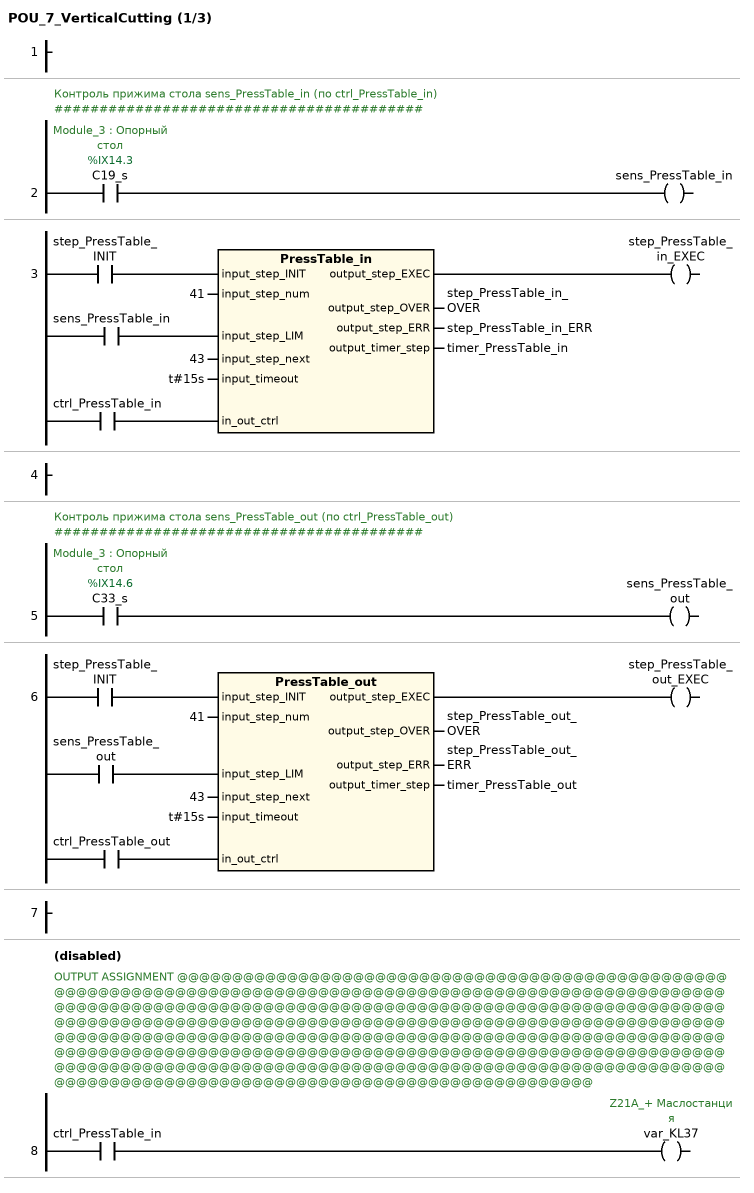
// NETWORK 1

// NETWORK 2
// Контроль прижима стола sens_PressTable_in (по ctrl_PressTable_in) #########################################
//   C19_s: Module_3 : Опорный стол | AT %IX14.3
sens_PressTable_in := C19_s;

// NETWORK 3
PressTable_in(input_step_INIT := step_PressTable_INIT, input_step_num := 41, input_step_LIM := sens_PressTable_in, input_step_next := 43, input_timeout := t#15s, in_out_ctrl := ctrl_PressTable_in, output_step_OVER => step_PressTable_in_OVER, output_step_ERR => step_PressTable_in_ERR, output_timer_step => timer_PressTable_in);
step_PressTable_in_EXEC := PressTable_in.output_step_EXEC;

// NETWORK 4

// NETWORK 5
// Контроль прижима стола sens_PressTable_out (по ctrl_PressTable_out) #########################################
//   C33_s: Module_3 : Опорный стол | AT %IX14.6
sens_PressTable_out := C33_s;

// NETWORK 6
PressTable_out(input_step_INIT := step_PressTable_INIT, input_step_num := 41, input_step_LIM := sens_PressTable_out, input_step_next := 43, input_timeout := t#15s, in_out_ctrl := ctrl_PressTable_out, output_step_OVER => step_PressTable_out_OVER, output_step_ERR => step_PressTable_out_ERR, output_timer_step => timer_PressTable_out);
step_PressTable_out_EXEC := PressTable_out.output_step_EXEC;

// NETWORK 7

// NETWORK 8 (disabled)
// OUTPUT ASSIGNMENT @@@@@@@@@@@@@@@@@@@@@@@@@@@@@@@@@@@@@@@@@@@@@@@@@@@@@@@@@@@@@@@@@@@@@@@@@@@@@@@@@@@@@@@@@@@@@@@@@@@@@@@@@@@@@@@@@@@@@@@@@@@@@@@@@@@@@@@@@@@@@@@@@@@@@@@@@@@@@@@@@@@@@@@@@@@@@@@@@@@@@@@@@@@@@@@@@@@@@@@@@@@@@@@@@@@@@@@@@@@@@@@@@@@@@@@@@@@@@@@@@@@@@@@@@@@@@@@@@@@@@@@@@@@@@@@@@@@@@@@@@@@@@@@@@@@@@@@@@@@@@@@@@@@@@@@@@@@@@@@@@@@@@@@@@@@@@@@@@@@@@@@@@@@@@@@@@@@@@@@@@@@@@@@@@@@@@@@@@@@@@@@@@@@@@@@@@@@@@@@@@@@@@@@@@@@@@@@@@@@@@@@@@@@@@@@@@@@@@@@@@@@@@@@@@@@@@@@@@@@@@@@@@
//   var_KL37: Z21A_+ Маслостанция
// var_KL37 := ctrl_PressTable_in;

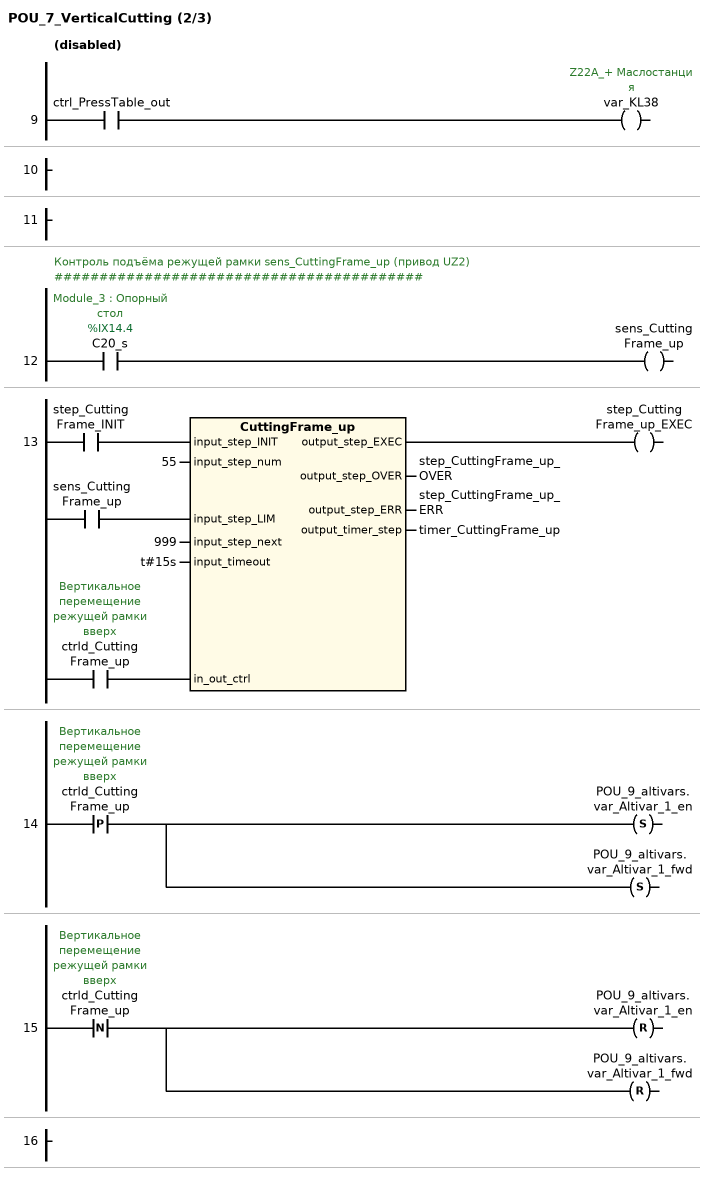
// NETWORK 9 (disabled)
//   var_KL38: Z22A_+ Маслостанция
// var_KL38 := ctrl_PressTable_out;

// NETWORK 10

// NETWORK 11

// NETWORK 12
// Контроль подъёма режущей рамки sens_CuttingFrame_up (привод UZ2) #########################################
//   C20_s: Module_3 : Опорный стол | AT %IX14.4
sens_CuttingFrame_up := C20_s;

// NETWORK 13
//   ctrld_CuttingFrame_up: Вертикальное перемещение режущей рамки вверх
CuttingFrame_up(input_step_INIT := step_CuttingFrame_INIT, input_step_num := 55, input_step_LIM := sens_CuttingFrame_up, input_step_next := 999, input_timeout := t#15s, in_out_ctrl := ctrld_CuttingFrame_up, output_step_OVER => step_CuttingFrame_up_OVER, output_step_ERR => step_CuttingFrame_up_ERR, output_timer_step => timer_CuttingFrame_up);
step_CuttingFrame_up_EXEC := CuttingFrame_up.output_step_EXEC;

// NETWORK 14
//   ctrld_CuttingFrame_up: Вертикальное перемещение режущей рамки вверх
_rt1(CLK := ctrld_CuttingFrame_up);
POU_9_altivars.var_Altivar_1_en S= _rt1.Q;
POU_9_altivars.var_Altivar_1_fwd S= _rt1.Q;

// NETWORK 15
//   ctrld_CuttingFrame_up: Вертикальное перемещение режущей рамки вверх
_ft1(CLK := ctrld_CuttingFrame_up);
POU_9_altivars.var_Altivar_1_en R= _ft1.Q;
POU_9_altivars.var_Altivar_1_fwd R= _ft1.Q;

// NETWORK 16

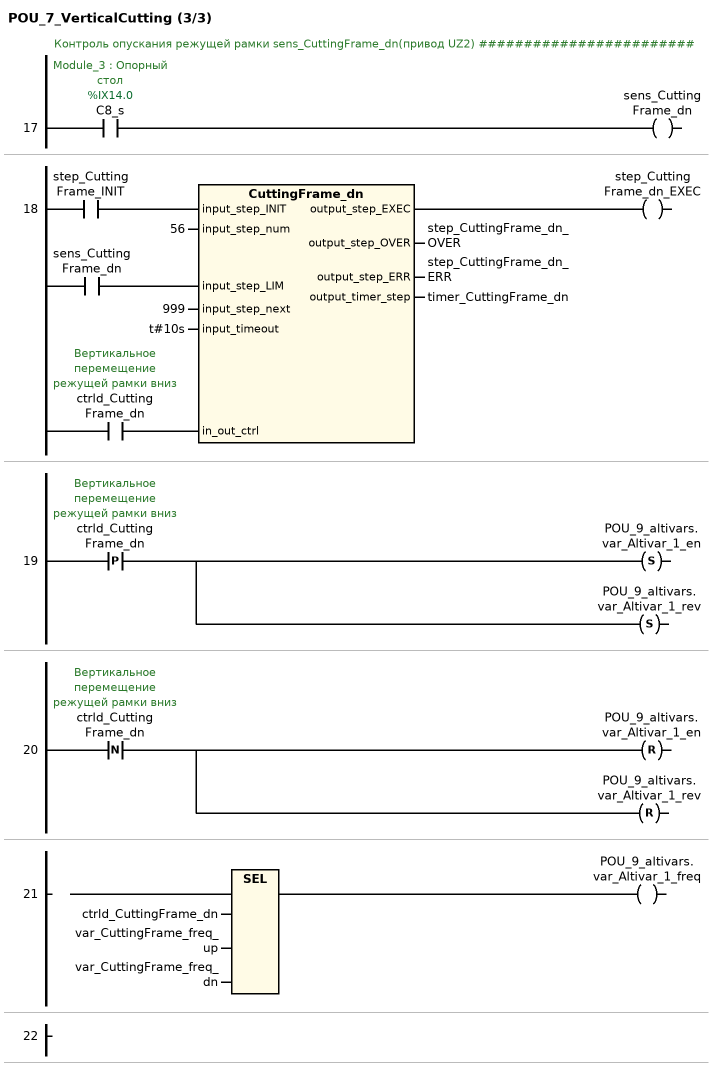
// NETWORK 17
// Контроль опускания режущей рамки sens_CuttingFrame_dn(привод UZ2) ########################
//   C8_s: Module_3 : Опорный стол | AT %IX14.0
sens_CuttingFrame_dn := C8_s;

// NETWORK 18
//   ctrld_CuttingFrame_dn: Вертикальное перемещение режущей рамки вниз
CuttingFrame_dn(input_step_INIT := step_CuttingFrame_INIT, input_step_num := 56, input_step_LIM := sens_CuttingFrame_dn, input_step_next := 999, input_timeout := t#10s, in_out_ctrl := ctrld_CuttingFrame_dn, output_step_OVER => step_CuttingFrame_dn_OVER, output_step_ERR => step_CuttingFrame_dn_ERR, output_timer_step => timer_CuttingFrame_dn);
step_CuttingFrame_dn_EXEC := CuttingFrame_dn.output_step_EXEC;

// NETWORK 19
//   ctrld_CuttingFrame_dn: Вертикальное перемещение режущей рамки вниз
_rt2(CLK := ctrld_CuttingFrame_dn);
POU_9_altivars.var_Altivar_1_en S= _rt2.Q;
POU_9_altivars.var_Altivar_1_rev S= _rt2.Q;

// NETWORK 20
//   ctrld_CuttingFrame_dn: Вертикальное перемещение режущей рамки вниз
_ft2(CLK := ctrld_CuttingFrame_dn);
POU_9_altivars.var_Altivar_1_en R= _ft2.Q;
POU_9_altivars.var_Altivar_1_rev R= _ft2.Q;

// NETWORK 21
//   ctrld_CuttingFrame_dn: Вертикальное перемещение режущей рамки вниз
POU_9_altivars.var_Altivar_1_freq := SEL(ctrld_CuttingFrame_dn, var_CuttingFrame_freq_up, var_CuttingFrame_freq_dn);

// NETWORK 22

END_PROGRAM

// MyController/Application/module_unites/PressTable_in
PROGRAM PressTable_in
VAR_INPUT
	input_step_INIT: BOOL;
	input_step_num: INT;
	input_step_LIM: BOOL;
	input_step_next: INT;
	input_timeout: TIME;
END_VAR

VAR_OUTPUT
	output_step_EXEC: BOOL;
	output_step_OVER: BOOL;
	output_step_ERR: BOOL;
	output_timer_step: TIME;
END_VAR
VAR_IN_OUT
	in_out_ctrl: BOOL;
END_VAR
VAR
	TON_step: TON;
	TON_step_res: BOOL;
	step_active: BOOL;
	TON_delay: TON;
	timer_delay: TIME;
	ton_delay_ok: BOOL;
END_VAR
VAR // added by the converter: edge detectors and wires of the graphical bodies
    _rt1, _rt2, _rt3, _rt4, _rt5, _rt6, _rt7 : R_TRIG;
    _w1, _w2 : BOOL;
    _ft1 : F_TRIG;
END_VAR

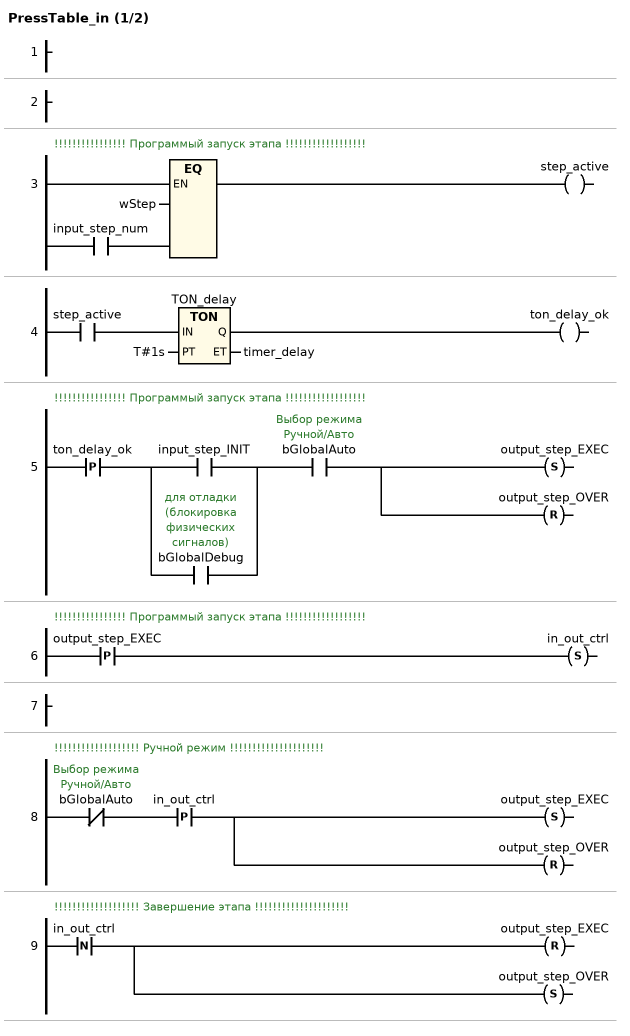
// NETWORK 1

// NETWORK 2

// NETWORK 3
// !!!!!!!!!!!!!!!! Программый запуск этапа !!!!!!!!!!!!!!!!!!
step_active := wStep = input_step_num;

// NETWORK 4
TON_delay(IN := step_active, PT := T#1s, ET => timer_delay); // TON
ton_delay_ok := TON_delay.Q;

// NETWORK 5
// !!!!!!!!!!!!!!!! Программый запуск этапа !!!!!!!!!!!!!!!!!!
//   bGlobalDebug: для отладки (блокировка физических сигналов)
//   bGlobalAuto: Выбор режима Ручной/Авто
_rt1(CLK := ton_delay_ok);
_w1 := _rt1.Q AND (input_step_INIT OR bGlobalDebug) AND bGlobalAuto;
output_step_EXEC S= _w1;
output_step_OVER R= _w1;

// NETWORK 6
// !!!!!!!!!!!!!!!! Программый запуск этапа !!!!!!!!!!!!!!!!!!
_rt2(CLK := output_step_EXEC);
in_out_ctrl S= _rt2.Q;

// NETWORK 7

// NETWORK 8
// !!!!!!!!!!!!!!!!!!! Ручной режим !!!!!!!!!!!!!!!!!!!!!
//   bGlobalAuto: Выбор режима Ручной/Авто
_rt3(CLK := in_out_ctrl);
_w2 := NOT bGlobalAuto AND _rt3.Q;
output_step_EXEC S= _w2;
output_step_OVER R= _w2;

// NETWORK 9
// !!!!!!!!!!!!!!!!!!! Завершение этапа !!!!!!!!!!!!!!!!!!!!!
_ft1(CLK := in_out_ctrl);
output_step_EXEC R= _ft1.Q;
output_step_OVER S= _ft1.Q;

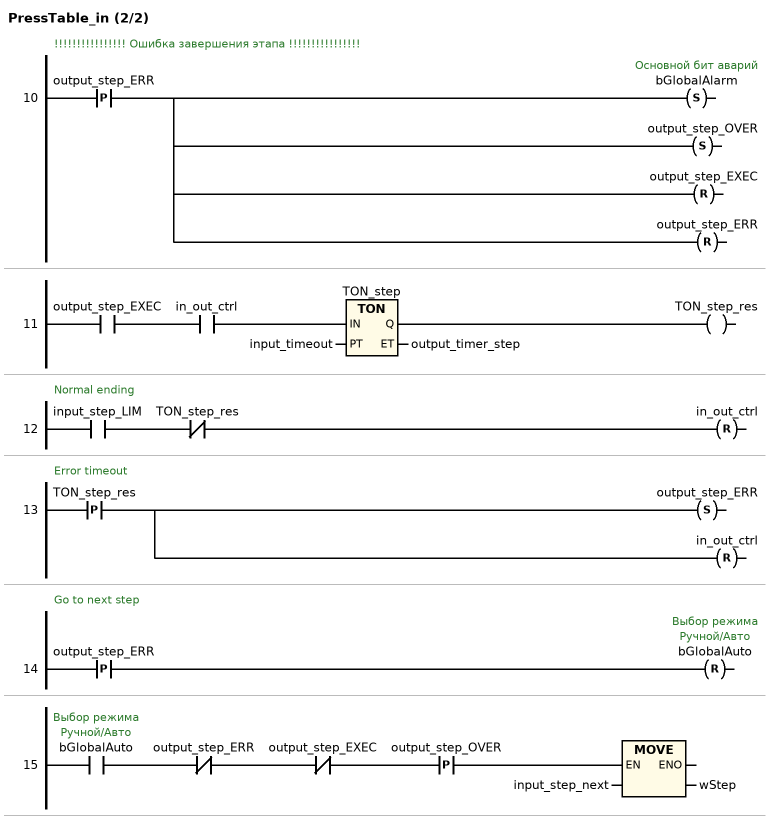
// NETWORK 10
// !!!!!!!!!!!!!!!! Ошибка завершения этапа !!!!!!!!!!!!!!!!
//   bGlobalAlarm: Основной бит аварий
_rt4(CLK := output_step_ERR);
bGlobalAlarm S= _rt4.Q;
output_step_OVER S= _rt4.Q;
output_step_EXEC R= _rt4.Q;
output_step_ERR R= _rt4.Q;

// NETWORK 11
TON_step(IN := output_step_EXEC AND in_out_ctrl, PT := input_timeout, ET => output_timer_step); // TON
TON_step_res := TON_step.Q;

// NETWORK 12
// Normal ending
in_out_ctrl R= input_step_LIM AND NOT TON_step_res;

// NETWORK 13
// Error timeout
_rt5(CLK := TON_step_res);
output_step_ERR S= _rt5.Q;
in_out_ctrl R= _rt5.Q;

// NETWORK 14
// Go to next step
//   bGlobalAuto: Выбор режима Ручной/Авто
_rt6(CLK := output_step_ERR);
bGlobalAuto R= _rt6.Q;

// NETWORK 15
//   bGlobalAuto: Выбор режима Ручной/Авто
_rt7(CLK := output_step_OVER);
IF bGlobalAuto AND NOT output_step_ERR AND NOT output_step_EXEC AND _rt7.Q THEN wStep := input_step_next; END_IF

END_PROGRAM

// MyController/Application/module_unites/PressTable_out
PROGRAM PressTable_out
VAR_INPUT
	input_step_INIT: BOOL;
	input_step_num: INT;
	input_step_LIM: BOOL;
	input_step_next: INT;
	input_timeout: TIME;
END_VAR

VAR_OUTPUT
	output_step_EXEC: BOOL;
	output_step_OVER: BOOL;
	output_step_ERR: BOOL;
	output_timer_step: TIME;
END_VAR
VAR_IN_OUT
	in_out_ctrl: BOOL;
END_VAR
VAR
	TON_step: TON;
	TON_step_res: BOOL;
	step_active: BOOL;
	TON_delay: TON;
	timer_delay: TIME;
	ton_delay_ok: BOOL;
END_VAR
VAR // added by the converter: edge detectors and wires of the graphical bodies
    _rt1, _rt2, _rt3, _rt4, _rt5, _rt6, _rt7 : R_TRIG;
    _w1, _w2 : BOOL;
    _ft1 : F_TRIG;
END_VAR

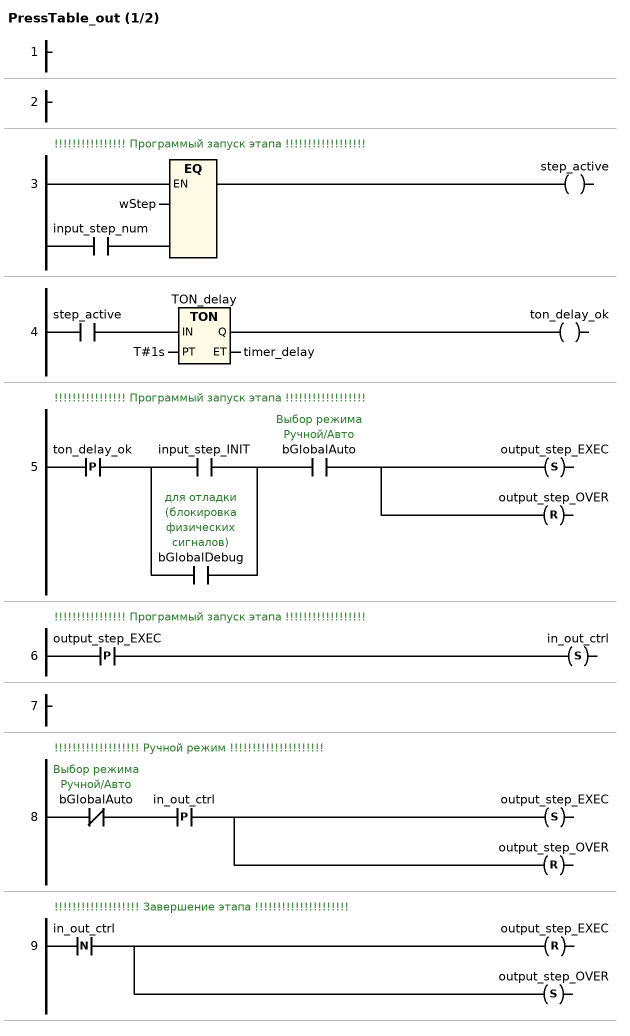
// NETWORK 1

// NETWORK 2

// NETWORK 3
// !!!!!!!!!!!!!!!! Программый запуск этапа !!!!!!!!!!!!!!!!!!
step_active := wStep = input_step_num;

// NETWORK 4
TON_delay(IN := step_active, PT := T#1s, ET => timer_delay); // TON
ton_delay_ok := TON_delay.Q;

// NETWORK 5
// !!!!!!!!!!!!!!!! Программый запуск этапа !!!!!!!!!!!!!!!!!!
//   bGlobalDebug: для отладки (блокировка физических сигналов)
//   bGlobalAuto: Выбор режима Ручной/Авто
_rt1(CLK := ton_delay_ok);
_w1 := _rt1.Q AND (input_step_INIT OR bGlobalDebug) AND bGlobalAuto;
output_step_EXEC S= _w1;
output_step_OVER R= _w1;

// NETWORK 6
// !!!!!!!!!!!!!!!! Программый запуск этапа !!!!!!!!!!!!!!!!!!
_rt2(CLK := output_step_EXEC);
in_out_ctrl S= _rt2.Q;

// NETWORK 7

// NETWORK 8
// !!!!!!!!!!!!!!!!!!! Ручной режим !!!!!!!!!!!!!!!!!!!!!
//   bGlobalAuto: Выбор режима Ручной/Авто
_rt3(CLK := in_out_ctrl);
_w2 := NOT bGlobalAuto AND _rt3.Q;
output_step_EXEC S= _w2;
output_step_OVER R= _w2;

// NETWORK 9
// !!!!!!!!!!!!!!!!!!! Завершение этапа !!!!!!!!!!!!!!!!!!!!!
_ft1(CLK := in_out_ctrl);
output_step_EXEC R= _ft1.Q;
output_step_OVER S= _ft1.Q;

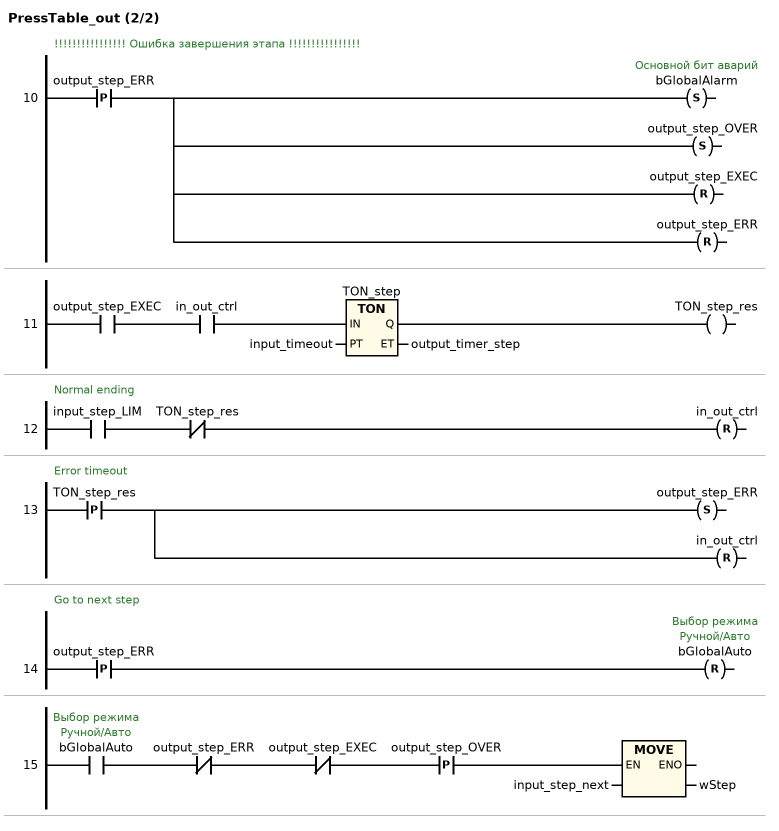
// NETWORK 10
// !!!!!!!!!!!!!!!! Ошибка завершения этапа !!!!!!!!!!!!!!!!
//   bGlobalAlarm: Основной бит аварий
_rt4(CLK := output_step_ERR);
bGlobalAlarm S= _rt4.Q;
output_step_OVER S= _rt4.Q;
output_step_EXEC R= _rt4.Q;
output_step_ERR R= _rt4.Q;

// NETWORK 11
TON_step(IN := output_step_EXEC AND in_out_ctrl, PT := input_timeout, ET => output_timer_step); // TON
TON_step_res := TON_step.Q;

// NETWORK 12
// Normal ending
in_out_ctrl R= input_step_LIM AND NOT TON_step_res;

// NETWORK 13
// Error timeout
_rt5(CLK := TON_step_res);
output_step_ERR S= _rt5.Q;
in_out_ctrl R= _rt5.Q;

// NETWORK 14
// Go to next step
//   bGlobalAuto: Выбор режима Ручной/Авто
_rt6(CLK := output_step_ERR);
bGlobalAuto R= _rt6.Q;

// NETWORK 15
//   bGlobalAuto: Выбор режима Ручной/Авто
_rt7(CLK := output_step_OVER);
IF bGlobalAuto AND NOT output_step_ERR AND NOT output_step_EXEC AND _rt7.Q THEN wStep := input_step_next; END_IF

END_PROGRAM

// MyController/Application/module_unites/CuttingFrame_up
PROGRAM CuttingFrame_up
VAR_INPUT
	input_step_INIT: BOOL;
	input_step_num: INT;
	input_step_LIM: BOOL;
	input_step_next: INT;
	input_timeout: TIME;
END_VAR

VAR_OUTPUT
	output_step_EXEC: BOOL;
	output_step_OVER: BOOL;
	output_step_ERR: BOOL;
	output_timer_step: TIME;
END_VAR
VAR_IN_OUT
	in_out_ctrl: BOOL;
END_VAR
VAR
	TON_step: TON;
	TON_step_res: BOOL;
	step_active: BOOL;
	TON_delay: TON;
	timer_delay: TIME;
	ton_delay_ok: BOOL;
END_VAR
VAR // added by the converter: edge detectors and wires of the graphical bodies
    _rt1, _rt2, _rt3, _rt4, _rt5, _rt6, _rt7 : R_TRIG;
    _w1, _w2 : BOOL;
    _ft1 : F_TRIG;
END_VAR

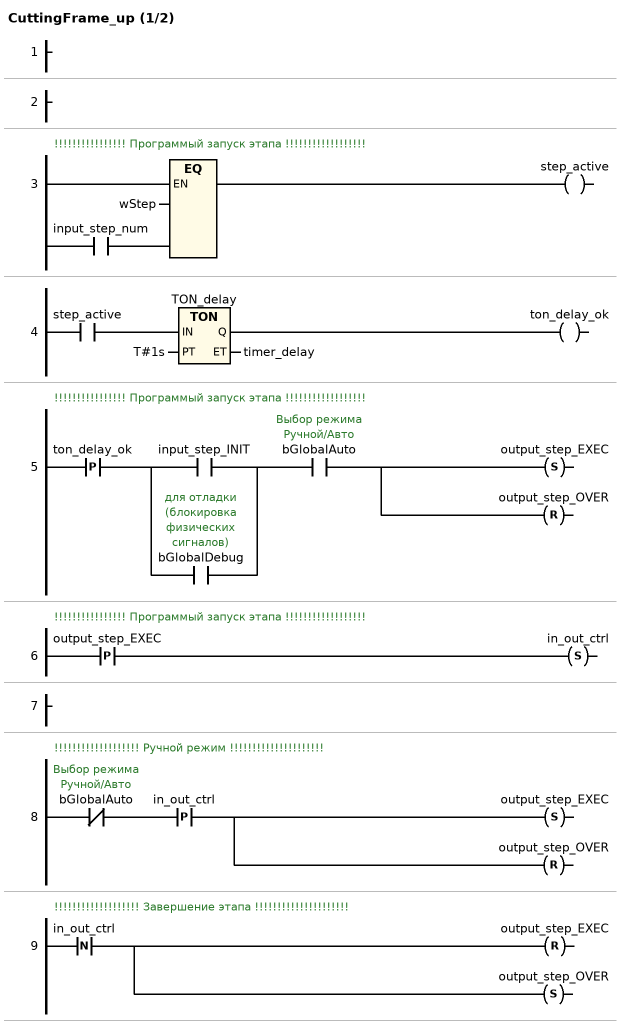
// NETWORK 1

// NETWORK 2

// NETWORK 3
// !!!!!!!!!!!!!!!! Программый запуск этапа !!!!!!!!!!!!!!!!!!
step_active := wStep = input_step_num;

// NETWORK 4
TON_delay(IN := step_active, PT := T#1s, ET => timer_delay); // TON
ton_delay_ok := TON_delay.Q;

// NETWORK 5
// !!!!!!!!!!!!!!!! Программый запуск этапа !!!!!!!!!!!!!!!!!!
//   bGlobalDebug: для отладки (блокировка физических сигналов)
//   bGlobalAuto: Выбор режима Ручной/Авто
_rt1(CLK := ton_delay_ok);
_w1 := _rt1.Q AND (input_step_INIT OR bGlobalDebug) AND bGlobalAuto;
output_step_EXEC S= _w1;
output_step_OVER R= _w1;

// NETWORK 6
// !!!!!!!!!!!!!!!! Программый запуск этапа !!!!!!!!!!!!!!!!!!
_rt2(CLK := output_step_EXEC);
in_out_ctrl S= _rt2.Q;

// NETWORK 7

// NETWORK 8
// !!!!!!!!!!!!!!!!!!! Ручной режим !!!!!!!!!!!!!!!!!!!!!
//   bGlobalAuto: Выбор режима Ручной/Авто
_rt3(CLK := in_out_ctrl);
_w2 := NOT bGlobalAuto AND _rt3.Q;
output_step_EXEC S= _w2;
output_step_OVER R= _w2;

// NETWORK 9
// !!!!!!!!!!!!!!!!!!! Завершение этапа !!!!!!!!!!!!!!!!!!!!!
_ft1(CLK := in_out_ctrl);
output_step_EXEC R= _ft1.Q;
output_step_OVER S= _ft1.Q;

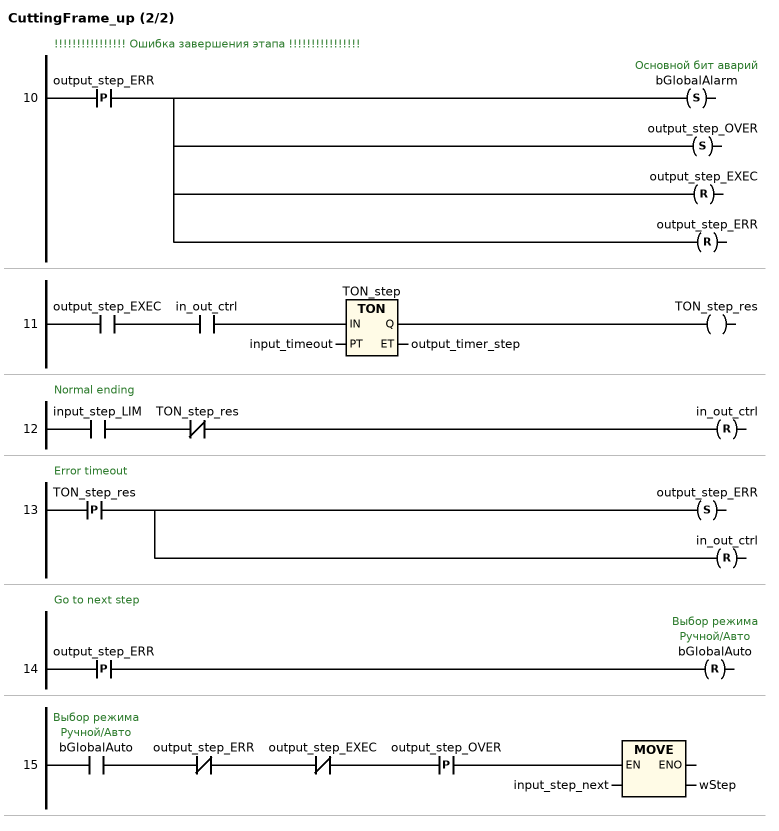
// NETWORK 10
// !!!!!!!!!!!!!!!! Ошибка завершения этапа !!!!!!!!!!!!!!!!
//   bGlobalAlarm: Основной бит аварий
_rt4(CLK := output_step_ERR);
bGlobalAlarm S= _rt4.Q;
output_step_OVER S= _rt4.Q;
output_step_EXEC R= _rt4.Q;
output_step_ERR R= _rt4.Q;

// NETWORK 11
TON_step(IN := output_step_EXEC AND in_out_ctrl, PT := input_timeout, ET => output_timer_step); // TON
TON_step_res := TON_step.Q;

// NETWORK 12
// Normal ending
in_out_ctrl R= input_step_LIM AND NOT TON_step_res;

// NETWORK 13
// Error timeout
_rt5(CLK := TON_step_res);
output_step_ERR S= _rt5.Q;
in_out_ctrl R= _rt5.Q;

// NETWORK 14
// Go to next step
//   bGlobalAuto: Выбор режима Ручной/Авто
_rt6(CLK := output_step_ERR);
bGlobalAuto R= _rt6.Q;

// NETWORK 15
//   bGlobalAuto: Выбор режима Ручной/Авто
_rt7(CLK := output_step_OVER);
IF bGlobalAuto AND NOT output_step_ERR AND NOT output_step_EXEC AND _rt7.Q THEN wStep := input_step_next; END_IF

END_PROGRAM

// MyController/Application/module_unites/CuttingFrame_dn
PROGRAM CuttingFrame_dn
VAR_INPUT
	input_step_INIT: BOOL;
	input_step_num: INT;
	input_step_LIM: BOOL;
	input_step_next: INT;
	input_timeout: TIME;
END_VAR

VAR_OUTPUT
	output_step_EXEC: BOOL;
	output_step_OVER: BOOL;
	output_step_ERR: BOOL;
	output_timer_step: TIME;
END_VAR
VAR_IN_OUT
	in_out_ctrl: BOOL;
END_VAR
VAR
	TON_step: TON;
	TON_step_res: BOOL;
	step_active: BOOL;
	TON_delay: TON;
	timer_delay: TIME;
	ton_delay_ok: BOOL;
END_VAR
VAR // added by the converter: edge detectors and wires of the graphical bodies
    _rt1, _rt2, _rt3, _rt4, _rt5, _rt6, _rt7 : R_TRIG;
    _w1, _w2 : BOOL;
    _ft1 : F_TRIG;
END_VAR

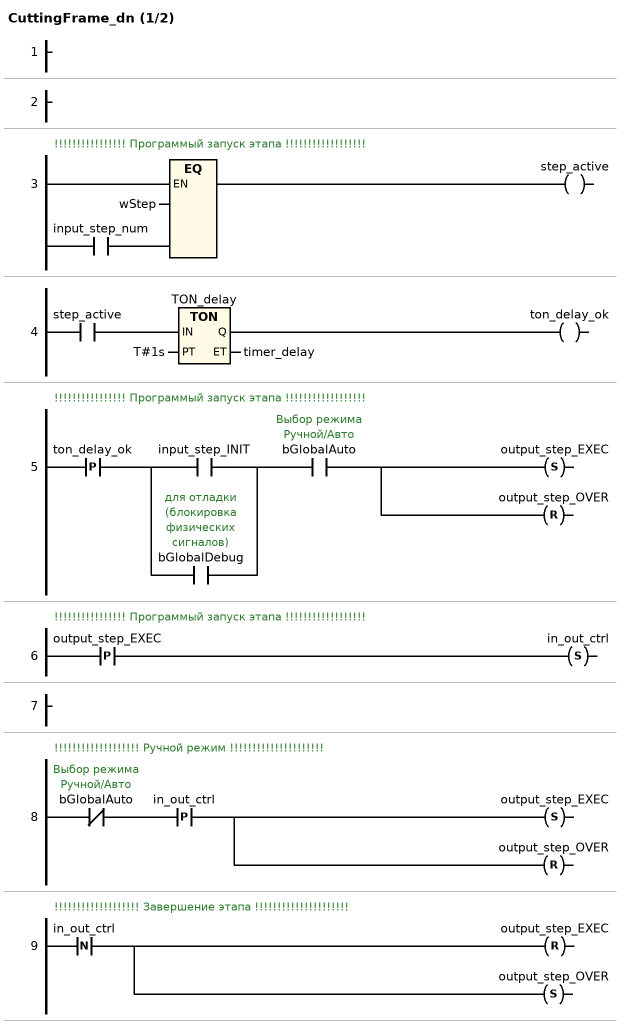
// NETWORK 1

// NETWORK 2

// NETWORK 3
// !!!!!!!!!!!!!!!! Программый запуск этапа !!!!!!!!!!!!!!!!!!
step_active := wStep = input_step_num;

// NETWORK 4
TON_delay(IN := step_active, PT := T#1s, ET => timer_delay); // TON
ton_delay_ok := TON_delay.Q;

// NETWORK 5
// !!!!!!!!!!!!!!!! Программый запуск этапа !!!!!!!!!!!!!!!!!!
//   bGlobalDebug: для отладки (блокировка физических сигналов)
//   bGlobalAuto: Выбор режима Ручной/Авто
_rt1(CLK := ton_delay_ok);
_w1 := _rt1.Q AND (input_step_INIT OR bGlobalDebug) AND bGlobalAuto;
output_step_EXEC S= _w1;
output_step_OVER R= _w1;

// NETWORK 6
// !!!!!!!!!!!!!!!! Программый запуск этапа !!!!!!!!!!!!!!!!!!
_rt2(CLK := output_step_EXEC);
in_out_ctrl S= _rt2.Q;

// NETWORK 7

// NETWORK 8
// !!!!!!!!!!!!!!!!!!! Ручной режим !!!!!!!!!!!!!!!!!!!!!
//   bGlobalAuto: Выбор режима Ручной/Авто
_rt3(CLK := in_out_ctrl);
_w2 := NOT bGlobalAuto AND _rt3.Q;
output_step_EXEC S= _w2;
output_step_OVER R= _w2;

// NETWORK 9
// !!!!!!!!!!!!!!!!!!! Завершение этапа !!!!!!!!!!!!!!!!!!!!!
_ft1(CLK := in_out_ctrl);
output_step_EXEC R= _ft1.Q;
output_step_OVER S= _ft1.Q;

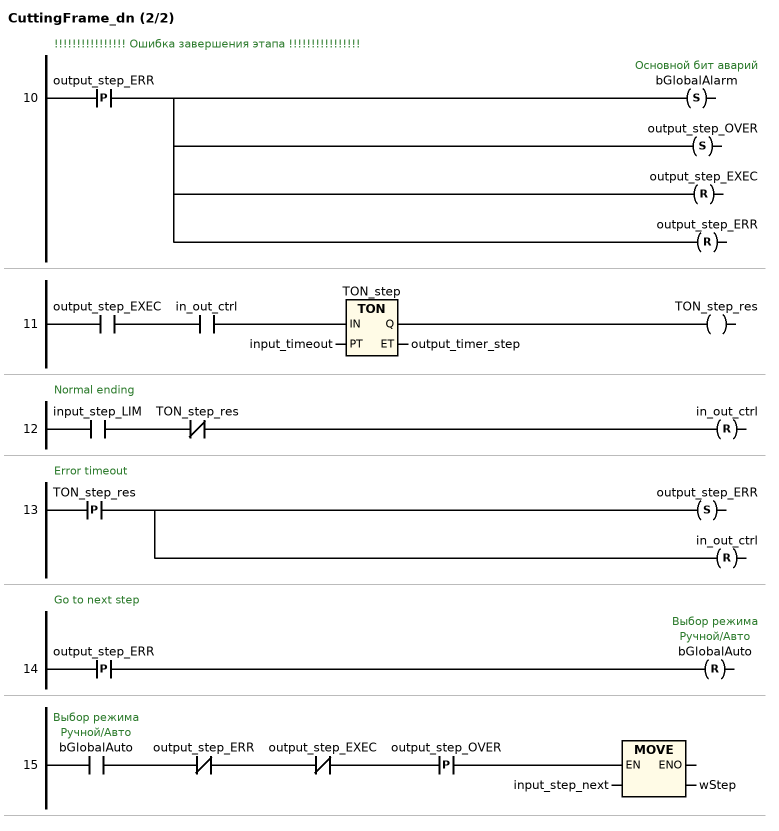
// NETWORK 10
// !!!!!!!!!!!!!!!! Ошибка завершения этапа !!!!!!!!!!!!!!!!
//   bGlobalAlarm: Основной бит аварий
_rt4(CLK := output_step_ERR);
bGlobalAlarm S= _rt4.Q;
output_step_OVER S= _rt4.Q;
output_step_EXEC R= _rt4.Q;
output_step_ERR R= _rt4.Q;

// NETWORK 11
TON_step(IN := output_step_EXEC AND in_out_ctrl, PT := input_timeout, ET => output_timer_step); // TON
TON_step_res := TON_step.Q;

// NETWORK 12
// Normal ending
in_out_ctrl R= input_step_LIM AND NOT TON_step_res;

// NETWORK 13
// Error timeout
_rt5(CLK := TON_step_res);
output_step_ERR S= _rt5.Q;
in_out_ctrl R= _rt5.Q;

// NETWORK 14
// Go to next step
//   bGlobalAuto: Выбор режима Ручной/Авто
_rt6(CLK := output_step_ERR);
bGlobalAuto R= _rt6.Q;

// NETWORK 15
//   bGlobalAuto: Выбор режима Ручной/Авто
_rt7(CLK := output_step_OVER);
IF bGlobalAuto AND NOT output_step_ERR AND NOT output_step_EXEC AND _rt7.Q THEN wStep := input_step_next; END_IF

END_PROGRAM

// MyController/Application/POU_5_Oprokidyvanie
PROGRAM POU_5_Oprokidyvanie
VAR
	sens_TakeTable_in: BOOL;
	ctrl_TakeTable_in: BOOL;
	step_TakeTable_INIT: BOOL := TRUE;
	step_TakeTable_in_EXEC: BOOL;
	step_TakeTable_in_OVER: BOOL;
	step_TakeTable_in_ERR: BOOL;
	timer_TakeTable_in: TIME;
	ctrl_TakeTable_out: BOOL;
	sens_TakeTable_out: BOOL;
	step_TakeTable_out_EXEC: BOOL;
	step_TakeTable_out_OVER: BOOL;
	step_TakeTable_out_ERR: BOOL;
	timer_TakeTable_out: TIME;
	ctrl_MoveTipper_in: BOOL;
	sens_MoveTipper_in: BOOL;
	step_MoveTipper_INIT: BOOL := TRUE;
	step_MoveTipper_in_EXEC: BOOL;
	step_MoveTipper_in_OVER: BOOL;
	step_MoveTipper_in_ERR: BOOL;
	timer_MoveTipper_in: TIME;
	ctrl_MoveTipper_out: BOOL;
	sens_MoveTipper_out: BOOL;
	step_MoveTipper_out_EXEC: BOOL;
	step_MoveTipper_out_OVER: BOOL;
	step_MoveTipper_out_ERR: BOOL;
	timer_MoveTipper_out: TIME;
	ctrl_FixingFrame_in: BOOL;
	sens_FixingFrame_in: BOOL;
	step_FixingFrame_INIT: BOOL := TRUE;
	step_FixingFrame_in_EXEC: BOOL;
	step_FixingFrame_in_OVER: BOOL;
	step_FixingFrame_in_ERR: BOOL;
	timer_FixingFrame_in: TIME;
	ctrl_FixingFrame_out: BOOL;
	sens_FixingFrame_out: BOOL;
	step_FixingFrame_out_EXEC: BOOL;
	step_FixingFrame_out_OVER: BOOL;
	step_FixingFrame_out_ERR: BOOL;
END_VAR

VAR
	timer_FixingFrame_out: TIME;
END_VAR

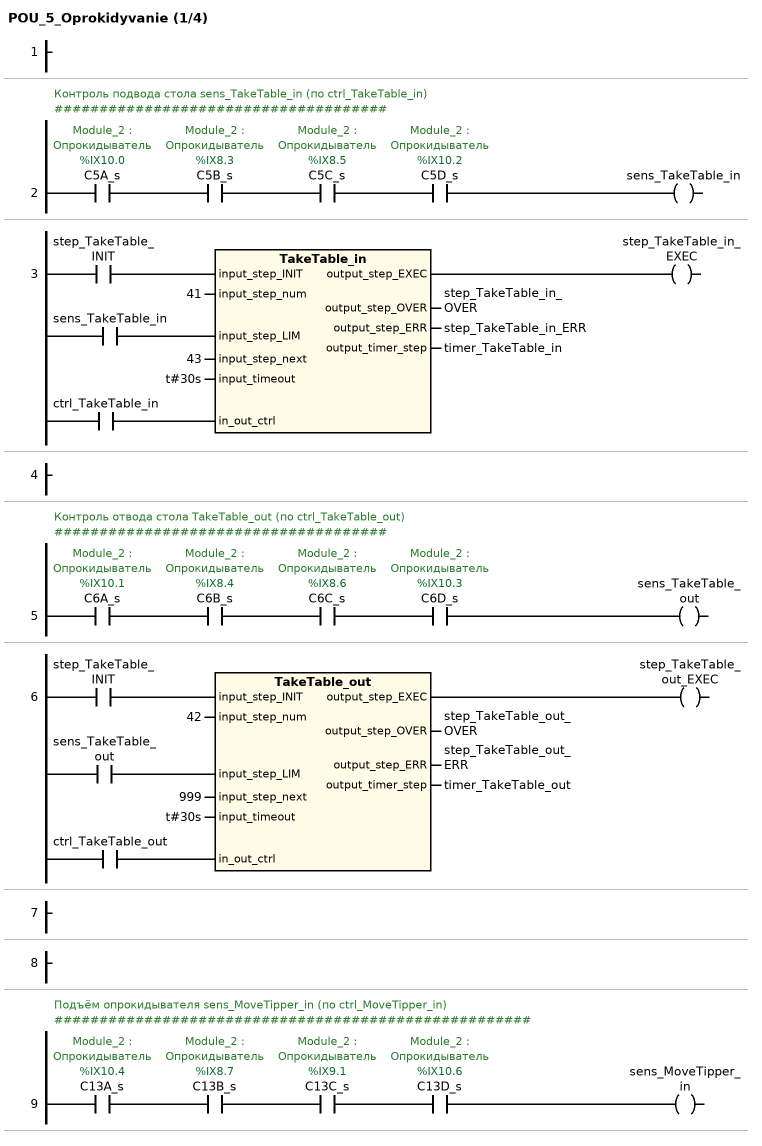
// NETWORK 1

// NETWORK 2
// Контроль подвода стола sens_TakeTable_in (по ctrl_TakeTable_in) #####################################
//   C5A_s: Module_2 : Опрокидыватель | AT %IX10.0
//   C5B_s: Module_2 : Опрокидыватель | AT %IX8.3
//   C5C_s: Module_2 : Опрокидыватель | AT %IX8.5
//   C5D_s: Module_2 : Опрокидыватель | AT %IX10.2
sens_TakeTable_in := C5A_s AND C5B_s AND C5C_s AND C5D_s;

// NETWORK 3
TakeTable_in(input_step_INIT := step_TakeTable_INIT, input_step_num := 41, input_step_LIM := sens_TakeTable_in, input_step_next := 43, input_timeout := t#30s, in_out_ctrl := ctrl_TakeTable_in, output_step_OVER => step_TakeTable_in_OVER, output_step_ERR => step_TakeTable_in_ERR, output_timer_step => timer_TakeTable_in);
step_TakeTable_in_EXEC := TakeTable_in.output_step_EXEC;

// NETWORK 4

// NETWORK 5
// Контроль отвода стола TakeTable_out (по ctrl_TakeTable_out) #####################################
//   C6A_s: Module_2 : Опрокидыватель | AT %IX10.1
//   C6B_s: Module_2 : Опрокидыватель | AT %IX8.4
//   C6C_s: Module_2 : Опрокидыватель | AT %IX8.6
//   C6D_s: Module_2 : Опрокидыватель | AT %IX10.3
sens_TakeTable_out := C6A_s AND C6B_s AND C6C_s AND C6D_s;

// NETWORK 6
TakeTable_out(input_step_INIT := step_TakeTable_INIT, input_step_num := 42, input_step_LIM := sens_TakeTable_out, input_step_next := 999, input_timeout := t#30s, in_out_ctrl := ctrl_TakeTable_out, output_step_OVER => step_TakeTable_out_OVER, output_step_ERR => step_TakeTable_out_ERR, output_timer_step => timer_TakeTable_out);
step_TakeTable_out_EXEC := TakeTable_out.output_step_EXEC;

// NETWORK 7

// NETWORK 8

// NETWORK 9
// Подъём опрокидывателя sens_MoveTipper_in (по ctrl_MoveTipper_in) #####################################################
//   C13A_s: Module_2 : Опрокидыватель | AT %IX10.4
//   C13B_s: Module_2 : Опрокидыватель | AT %IX8.7
//   C13C_s: Module_2 : Опрокидыватель | AT %IX9.1
//   C13D_s: Module_2 : Опрокидыватель | AT %IX10.6
sens_MoveTipper_in := C13A_s AND C13B_s AND C13C_s AND C13D_s;

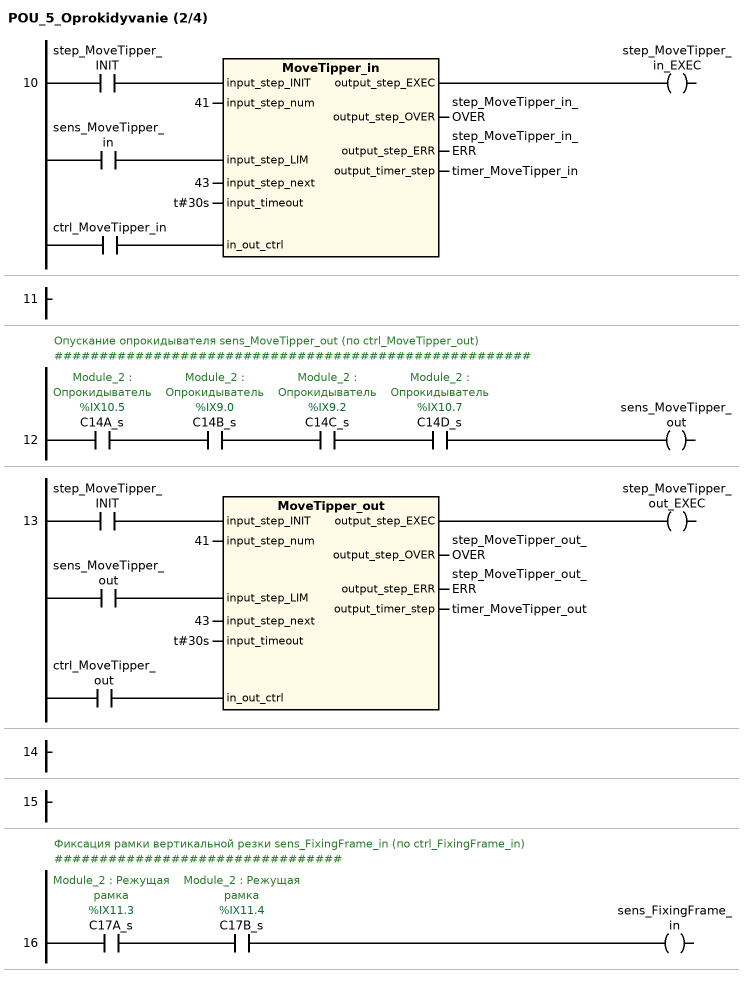
// NETWORK 10
MoveTipper_in(input_step_INIT := step_MoveTipper_INIT, input_step_num := 41, input_step_LIM := sens_MoveTipper_in, input_step_next := 43, input_timeout := t#30s, in_out_ctrl := ctrl_MoveTipper_in, output_step_OVER => step_MoveTipper_in_OVER, output_step_ERR => step_MoveTipper_in_ERR, output_timer_step => timer_MoveTipper_in);
step_MoveTipper_in_EXEC := MoveTipper_in.output_step_EXEC;

// NETWORK 11

// NETWORK 12
// Опускание опрокидывателя sens_MoveTipper_out (по ctrl_MoveTipper_out) #####################################################
//   C14A_s: Module_2 : Опрокидыватель | AT %IX10.5
//   C14B_s: Module_2 : Опрокидыватель | AT %IX9.0
//   C14C_s: Module_2 : Опрокидыватель | AT %IX9.2
//   C14D_s: Module_2 : Опрокидыватель | AT %IX10.7
sens_MoveTipper_out := C14A_s AND C14B_s AND C14C_s AND C14D_s;

// NETWORK 13
MoveTipper_out(input_step_INIT := step_MoveTipper_INIT, input_step_num := 41, input_step_LIM := sens_MoveTipper_out, input_step_next := 43, input_timeout := t#30s, in_out_ctrl := ctrl_MoveTipper_out, output_step_OVER => step_MoveTipper_out_OVER, output_step_ERR => step_MoveTipper_out_ERR, output_timer_step => timer_MoveTipper_out);
step_MoveTipper_out_EXEC := MoveTipper_out.output_step_EXEC;

// NETWORK 14

// NETWORK 15

// NETWORK 16
// Фиксация рамки вертикальной резки sens_FixingFrame_in (по ctrl_FixingFrame_in) ################################
//   C17A_s: Module_2 : Режущая рамка | AT %IX11.3
//   C17B_s: Module_2 : Режущая рамка | AT %IX11.4
sens_FixingFrame_in := C17A_s AND C17B_s;

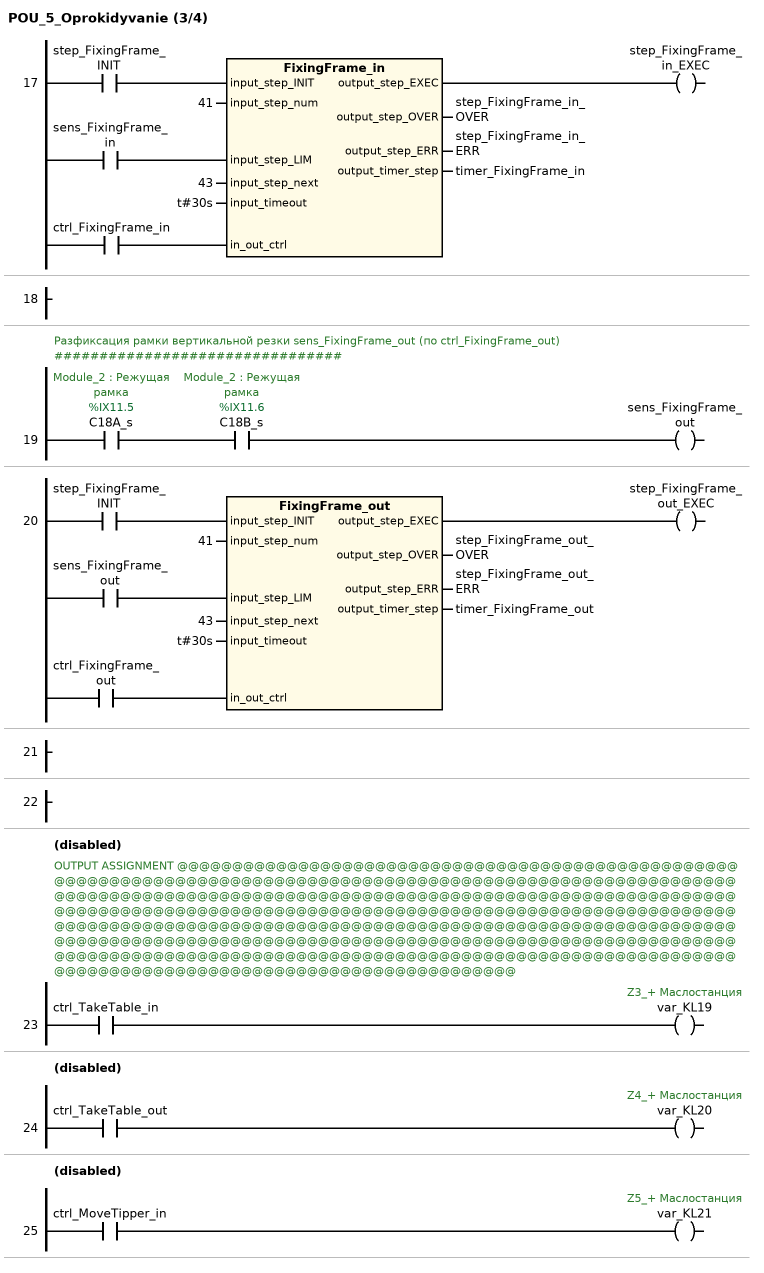
// NETWORK 17
FixingFrame_in(input_step_INIT := step_FixingFrame_INIT, input_step_num := 41, input_step_LIM := sens_FixingFrame_in, input_step_next := 43, input_timeout := t#30s, in_out_ctrl := ctrl_FixingFrame_in, output_step_OVER => step_FixingFrame_in_OVER, output_step_ERR => step_FixingFrame_in_ERR, output_timer_step => timer_FixingFrame_in);
step_FixingFrame_in_EXEC := FixingFrame_in.output_step_EXEC;

// NETWORK 18

// NETWORK 19
// Разфиксация рамки вертикальной резки sens_FixingFrame_out (по ctrl_FixingFrame_out) ################################
//   C18A_s: Module_2 : Режущая рамка | AT %IX11.5
//   C18B_s: Module_2 : Режущая рамка | AT %IX11.6
sens_FixingFrame_out := C18A_s AND C18B_s;

// NETWORK 20
FixingFrame_out(input_step_INIT := step_FixingFrame_INIT, input_step_num := 41, input_step_LIM := sens_FixingFrame_out, input_step_next := 43, input_timeout := t#30s, in_out_ctrl := ctrl_FixingFrame_out, output_step_OVER => step_FixingFrame_out_OVER, output_step_ERR => step_FixingFrame_out_ERR, output_timer_step => timer_FixingFrame_out);
step_FixingFrame_out_EXEC := FixingFrame_out.output_step_EXEC;

// NETWORK 21

// NETWORK 22

// NETWORK 23 (disabled)
// OUTPUT ASSIGNMENT @@@@@@@@@@@@@@@@@@@@@@@@@@@@@@@@@@@@@@@@@@@@@@@@@@@@@@@@@@@@@@@@@@@@@@@@@@@@@@@@@@@@@@@@@@@@@@@@@@@@@@@@@@@@@@@@@@@@@@@@@@@@@@@@@@@@@@@@@@@@@@@@@@@@@@@@@@@@@@@@@@@@@@@@@@@@@@@@@@@@@@@@@@@@@@@@@@@@@@@@@@@@@@@@@@@@@@@@@@@@@@@@@@@@@@@@@@@@@@@@@@@@@@@@@@@@@@@@@@@@@@@@@@@@@@@@@@@@@@@@@@@@@@@@@@@@@@@@@@@@@@@@@@@@@@@@@@@@@@@@@@@@@@@@@@@@@@@@@@@@@@@@@@@@@@@@@@@@@@@@@@@@@@@@@@@@@@@@@@@@@@@@@@@@@@@@@@@@@@@@@@@@@@@@@@@@@@@@@@@@@@@@@@@@@@@@@@@@@@@@@@@@@@@@@@@@@@@@@@@@@@@@@
//   var_KL19: Z3_+ Маслостанция
// var_KL19 := ctrl_TakeTable_in;

// NETWORK 24 (disabled)
//   var_KL20: Z4_+ Маслостанция
// var_KL20 := ctrl_TakeTable_out;

// NETWORK 25 (disabled)
//   var_KL21: Z5_+ Маслостанция
// var_KL21 := ctrl_MoveTipper_in;

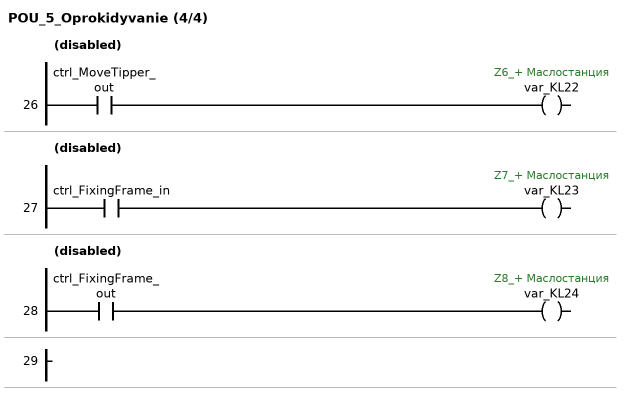
// NETWORK 26 (disabled)
//   var_KL22: Z6_+ Маслостанция
// var_KL22 := ctrl_MoveTipper_out;

// NETWORK 27 (disabled)
//   var_KL23: Z7_+ Маслостанция
// var_KL23 := ctrl_FixingFrame_in;

// NETWORK 28 (disabled)
//   var_KL24: Z8_+ Маслостанция
// var_KL24 := ctrl_FixingFrame_out;

// NETWORK 29

END_PROGRAM

// MyController/Application/module_unites/TakeTable_in
PROGRAM TakeTable_in
VAR_INPUT
	input_step_INIT: BOOL;
	input_step_num: INT;
	input_step_LIM: BOOL;
	input_step_next: INT;
	input_timeout: TIME;
END_VAR

VAR_OUTPUT
	output_step_EXEC: BOOL;
	output_step_OVER: BOOL;
	output_step_ERR: BOOL;
	output_timer_step: TIME;
END_VAR
VAR_IN_OUT
	in_out_ctrl: BOOL;
END_VAR
VAR
	TON_step: TON;
	TON_step_res: BOOL;
	step_active: BOOL;
	TON_delay: TON;
	timer_delay: TIME;
	ton_delay_ok: BOOL;
END_VAR
VAR // added by the converter: edge detectors and wires of the graphical bodies
    _rt1, _rt2, _rt3, _rt4, _rt5, _rt6, _rt7 : R_TRIG;
    _w1, _w2 : BOOL;
    _ft1 : F_TRIG;
END_VAR

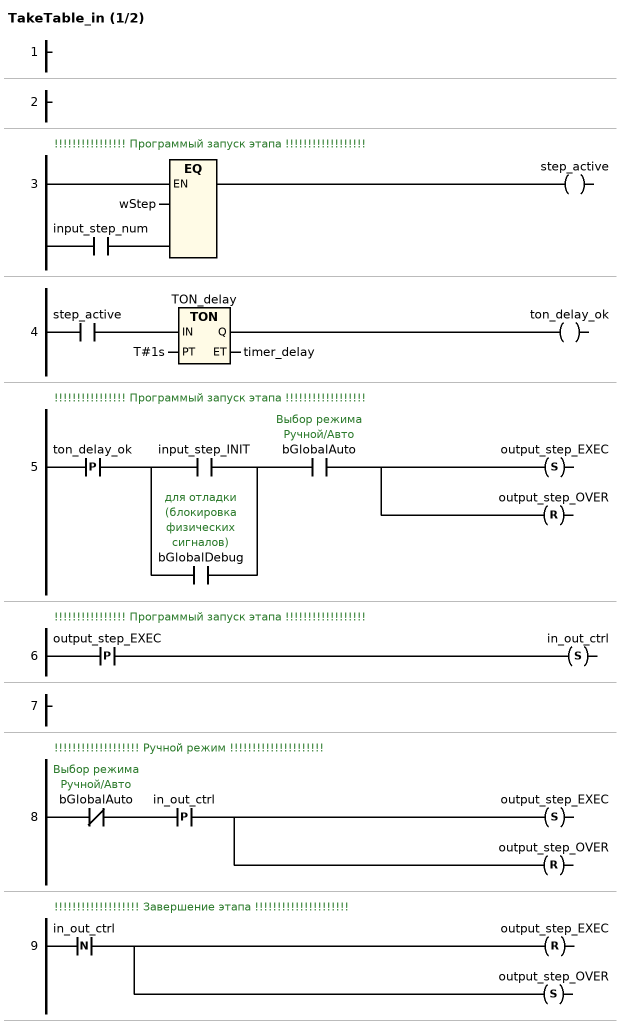
// NETWORK 1

// NETWORK 2

// NETWORK 3
// !!!!!!!!!!!!!!!! Программый запуск этапа !!!!!!!!!!!!!!!!!!
step_active := wStep = input_step_num;

// NETWORK 4
TON_delay(IN := step_active, PT := T#1s, ET => timer_delay); // TON
ton_delay_ok := TON_delay.Q;

// NETWORK 5
// !!!!!!!!!!!!!!!! Программый запуск этапа !!!!!!!!!!!!!!!!!!
//   bGlobalDebug: для отладки (блокировка физических сигналов)
//   bGlobalAuto: Выбор режима Ручной/Авто
_rt1(CLK := ton_delay_ok);
_w1 := _rt1.Q AND (input_step_INIT OR bGlobalDebug) AND bGlobalAuto;
output_step_EXEC S= _w1;
output_step_OVER R= _w1;

// NETWORK 6
// !!!!!!!!!!!!!!!! Программый запуск этапа !!!!!!!!!!!!!!!!!!
_rt2(CLK := output_step_EXEC);
in_out_ctrl S= _rt2.Q;

// NETWORK 7

// NETWORK 8
// !!!!!!!!!!!!!!!!!!! Ручной режим !!!!!!!!!!!!!!!!!!!!!
//   bGlobalAuto: Выбор режима Ручной/Авто
_rt3(CLK := in_out_ctrl);
_w2 := NOT bGlobalAuto AND _rt3.Q;
output_step_EXEC S= _w2;
output_step_OVER R= _w2;

// NETWORK 9
// !!!!!!!!!!!!!!!!!!! Завершение этапа !!!!!!!!!!!!!!!!!!!!!
_ft1(CLK := in_out_ctrl);
output_step_EXEC R= _ft1.Q;
output_step_OVER S= _ft1.Q;

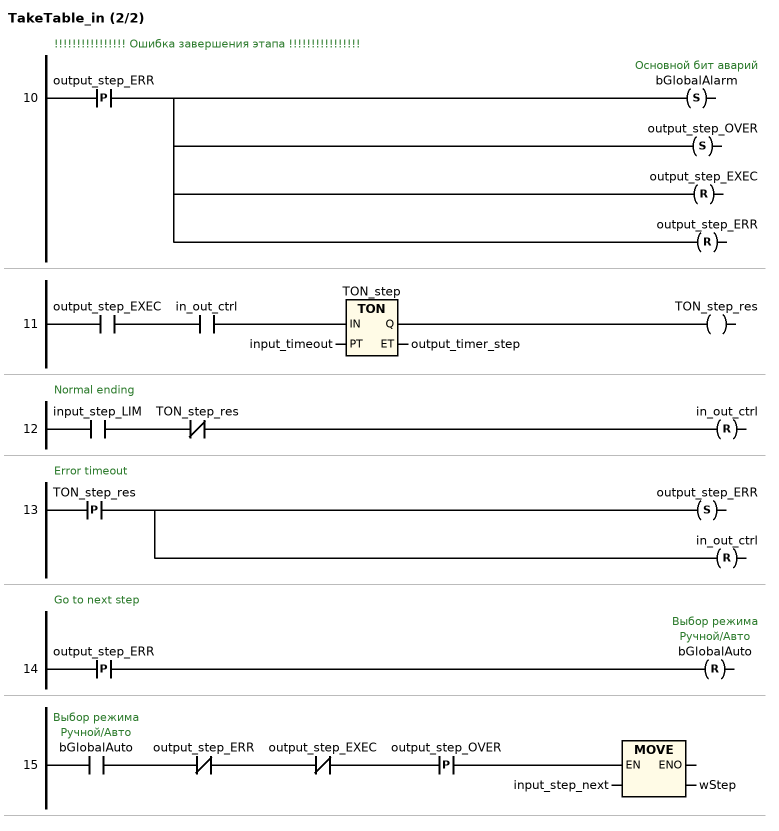
// NETWORK 10
// !!!!!!!!!!!!!!!! Ошибка завершения этапа !!!!!!!!!!!!!!!!
//   bGlobalAlarm: Основной бит аварий
_rt4(CLK := output_step_ERR);
bGlobalAlarm S= _rt4.Q;
output_step_OVER S= _rt4.Q;
output_step_EXEC R= _rt4.Q;
output_step_ERR R= _rt4.Q;

// NETWORK 11
TON_step(IN := output_step_EXEC AND in_out_ctrl, PT := input_timeout, ET => output_timer_step); // TON
TON_step_res := TON_step.Q;

// NETWORK 12
// Normal ending
in_out_ctrl R= input_step_LIM AND NOT TON_step_res;

// NETWORK 13
// Error timeout
_rt5(CLK := TON_step_res);
output_step_ERR S= _rt5.Q;
in_out_ctrl R= _rt5.Q;

// NETWORK 14
// Go to next step
//   bGlobalAuto: Выбор режима Ручной/Авто
_rt6(CLK := output_step_ERR);
bGlobalAuto R= _rt6.Q;

// NETWORK 15
//   bGlobalAuto: Выбор режима Ручной/Авто
_rt7(CLK := output_step_OVER);
IF bGlobalAuto AND NOT output_step_ERR AND NOT output_step_EXEC AND _rt7.Q THEN wStep := input_step_next; END_IF

END_PROGRAM

// MyController/Application/module_unites/TakeTable_out
PROGRAM TakeTable_out
VAR_INPUT
	input_step_INIT: BOOL;
	input_step_num: INT;
	input_step_LIM: BOOL;
	input_step_next: INT;
	input_timeout: TIME;
END_VAR

VAR_OUTPUT
	output_step_EXEC: BOOL;
	output_step_OVER: BOOL;
	output_step_ERR: BOOL;
	output_timer_step: TIME;
END_VAR
VAR_IN_OUT
	in_out_ctrl: BOOL;
END_VAR
VAR
	TON_step: TON;
	TON_step_res: BOOL;
	step_active: BOOL;
	TON_delay: TON;
	timer_delay: TIME;
	ton_delay_ok: BOOL;
END_VAR
VAR // added by the converter: edge detectors and wires of the graphical bodies
    _rt1, _rt2, _rt3, _rt4, _rt5, _rt6, _rt7 : R_TRIG;
    _w1, _w2 : BOOL;
    _ft1 : F_TRIG;
END_VAR

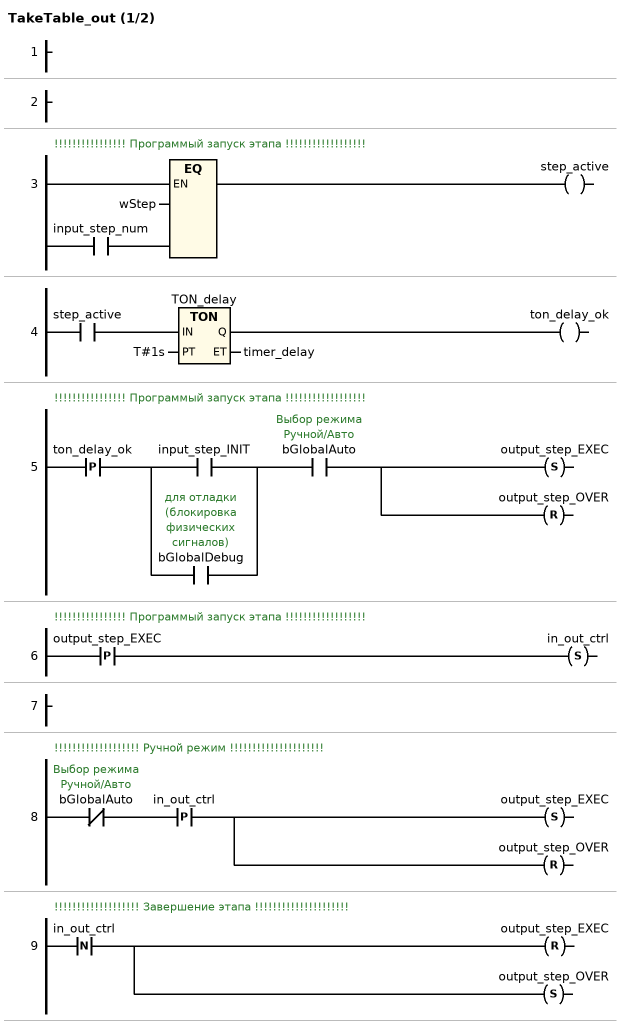
// NETWORK 1

// NETWORK 2

// NETWORK 3
// !!!!!!!!!!!!!!!! Программый запуск этапа !!!!!!!!!!!!!!!!!!
step_active := wStep = input_step_num;

// NETWORK 4
TON_delay(IN := step_active, PT := T#1s, ET => timer_delay); // TON
ton_delay_ok := TON_delay.Q;

// NETWORK 5
// !!!!!!!!!!!!!!!! Программый запуск этапа !!!!!!!!!!!!!!!!!!
//   bGlobalDebug: для отладки (блокировка физических сигналов)
//   bGlobalAuto: Выбор режима Ручной/Авто
_rt1(CLK := ton_delay_ok);
_w1 := _rt1.Q AND (input_step_INIT OR bGlobalDebug) AND bGlobalAuto;
output_step_EXEC S= _w1;
output_step_OVER R= _w1;

// NETWORK 6
// !!!!!!!!!!!!!!!! Программый запуск этапа !!!!!!!!!!!!!!!!!!
_rt2(CLK := output_step_EXEC);
in_out_ctrl S= _rt2.Q;

// NETWORK 7

// NETWORK 8
// !!!!!!!!!!!!!!!!!!! Ручной режим !!!!!!!!!!!!!!!!!!!!!
//   bGlobalAuto: Выбор режима Ручной/Авто
_rt3(CLK := in_out_ctrl);
_w2 := NOT bGlobalAuto AND _rt3.Q;
output_step_EXEC S= _w2;
output_step_OVER R= _w2;

// NETWORK 9
// !!!!!!!!!!!!!!!!!!! Завершение этапа !!!!!!!!!!!!!!!!!!!!!
_ft1(CLK := in_out_ctrl);
output_step_EXEC R= _ft1.Q;
output_step_OVER S= _ft1.Q;

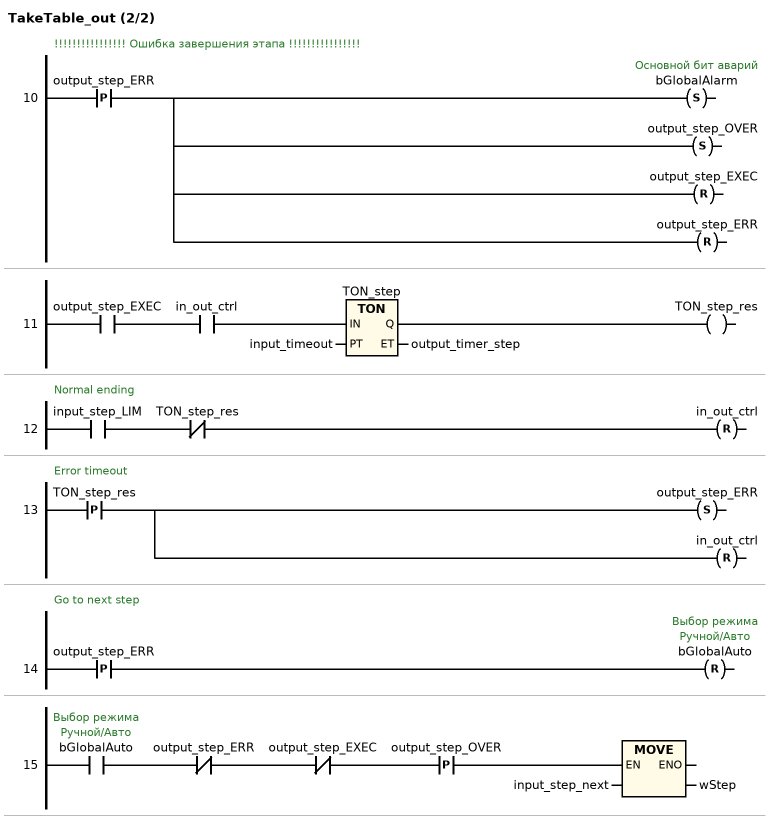
// NETWORK 10
// !!!!!!!!!!!!!!!! Ошибка завершения этапа !!!!!!!!!!!!!!!!
//   bGlobalAlarm: Основной бит аварий
_rt4(CLK := output_step_ERR);
bGlobalAlarm S= _rt4.Q;
output_step_OVER S= _rt4.Q;
output_step_EXEC R= _rt4.Q;
output_step_ERR R= _rt4.Q;

// NETWORK 11
TON_step(IN := output_step_EXEC AND in_out_ctrl, PT := input_timeout, ET => output_timer_step); // TON
TON_step_res := TON_step.Q;

// NETWORK 12
// Normal ending
in_out_ctrl R= input_step_LIM AND NOT TON_step_res;

// NETWORK 13
// Error timeout
_rt5(CLK := TON_step_res);
output_step_ERR S= _rt5.Q;
in_out_ctrl R= _rt5.Q;

// NETWORK 14
// Go to next step
//   bGlobalAuto: Выбор режима Ручной/Авто
_rt6(CLK := output_step_ERR);
bGlobalAuto R= _rt6.Q;

// NETWORK 15
//   bGlobalAuto: Выбор режима Ручной/Авто
_rt7(CLK := output_step_OVER);
IF bGlobalAuto AND NOT output_step_ERR AND NOT output_step_EXEC AND _rt7.Q THEN wStep := input_step_next; END_IF

END_PROGRAM

// MyController/Application/module_unites/MoveTipper_in
PROGRAM MoveTipper_in
VAR_INPUT
	input_step_INIT: BOOL;
	input_step_num: INT;
	input_step_LIM: BOOL;
	input_step_next: INT;
	input_timeout: TIME;
END_VAR

VAR_OUTPUT
	output_step_EXEC: BOOL;
	output_step_OVER: BOOL;
	output_step_ERR: BOOL;
	output_timer_step: TIME;
END_VAR
VAR_IN_OUT
	in_out_ctrl: BOOL;
END_VAR
VAR
	TON_step: TON;
	TON_step_res: BOOL;
	step_active: BOOL;
	TON_delay: TON;
	timer_delay: TIME;
	ton_delay_ok: BOOL;
END_VAR
VAR // added by the converter: edge detectors and wires of the graphical bodies
    _rt1, _rt2, _rt3, _rt4, _rt5, _rt6, _rt7 : R_TRIG;
    _w1, _w2 : BOOL;
    _ft1 : F_TRIG;
END_VAR

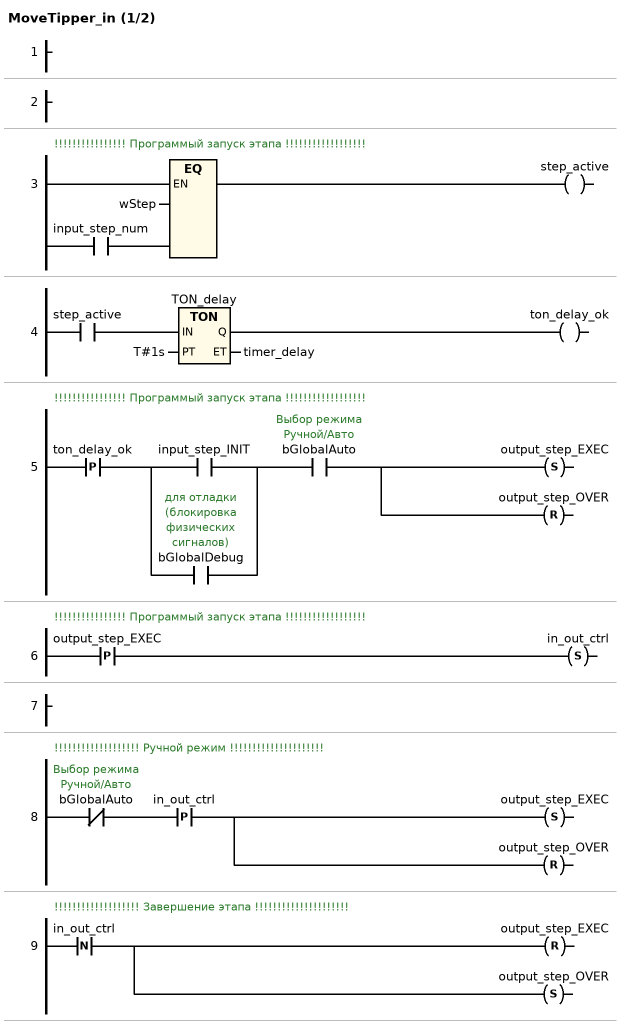
// NETWORK 1

// NETWORK 2

// NETWORK 3
// !!!!!!!!!!!!!!!! Программый запуск этапа !!!!!!!!!!!!!!!!!!
step_active := wStep = input_step_num;

// NETWORK 4
TON_delay(IN := step_active, PT := T#1s, ET => timer_delay); // TON
ton_delay_ok := TON_delay.Q;

// NETWORK 5
// !!!!!!!!!!!!!!!! Программый запуск этапа !!!!!!!!!!!!!!!!!!
//   bGlobalDebug: для отладки (блокировка физических сигналов)
//   bGlobalAuto: Выбор режима Ручной/Авто
_rt1(CLK := ton_delay_ok);
_w1 := _rt1.Q AND (input_step_INIT OR bGlobalDebug) AND bGlobalAuto;
output_step_EXEC S= _w1;
output_step_OVER R= _w1;

// NETWORK 6
// !!!!!!!!!!!!!!!! Программый запуск этапа !!!!!!!!!!!!!!!!!!
_rt2(CLK := output_step_EXEC);
in_out_ctrl S= _rt2.Q;

// NETWORK 7

// NETWORK 8
// !!!!!!!!!!!!!!!!!!! Ручной режим !!!!!!!!!!!!!!!!!!!!!
//   bGlobalAuto: Выбор режима Ручной/Авто
_rt3(CLK := in_out_ctrl);
_w2 := NOT bGlobalAuto AND _rt3.Q;
output_step_EXEC S= _w2;
output_step_OVER R= _w2;

// NETWORK 9
// !!!!!!!!!!!!!!!!!!! Завершение этапа !!!!!!!!!!!!!!!!!!!!!
_ft1(CLK := in_out_ctrl);
output_step_EXEC R= _ft1.Q;
output_step_OVER S= _ft1.Q;

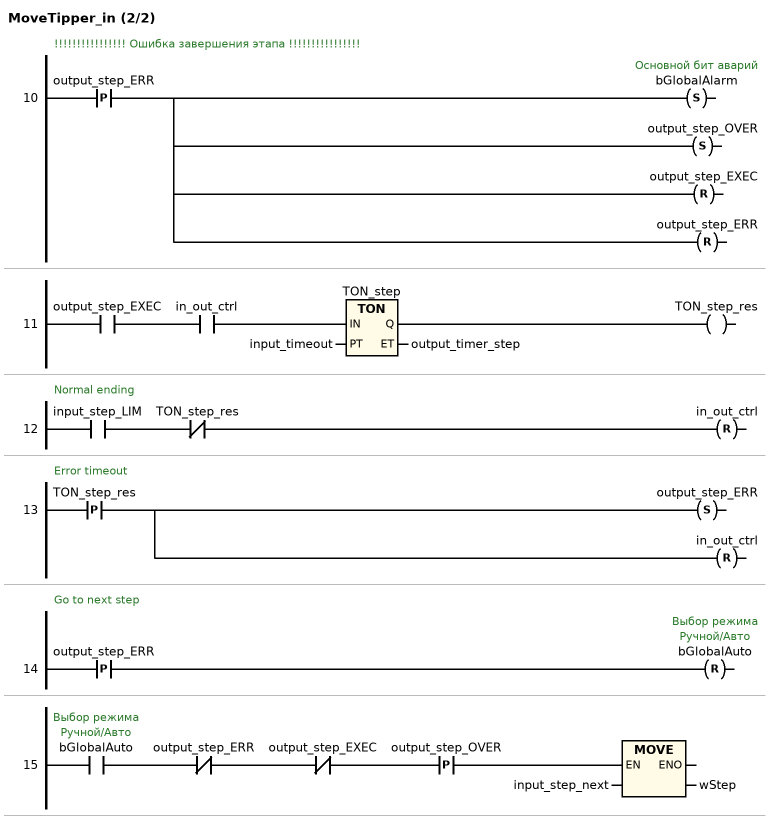
// NETWORK 10
// !!!!!!!!!!!!!!!! Ошибка завершения этапа !!!!!!!!!!!!!!!!
//   bGlobalAlarm: Основной бит аварий
_rt4(CLK := output_step_ERR);
bGlobalAlarm S= _rt4.Q;
output_step_OVER S= _rt4.Q;
output_step_EXEC R= _rt4.Q;
output_step_ERR R= _rt4.Q;

// NETWORK 11
TON_step(IN := output_step_EXEC AND in_out_ctrl, PT := input_timeout, ET => output_timer_step); // TON
TON_step_res := TON_step.Q;

// NETWORK 12
// Normal ending
in_out_ctrl R= input_step_LIM AND NOT TON_step_res;

// NETWORK 13
// Error timeout
_rt5(CLK := TON_step_res);
output_step_ERR S= _rt5.Q;
in_out_ctrl R= _rt5.Q;

// NETWORK 14
// Go to next step
//   bGlobalAuto: Выбор режима Ручной/Авто
_rt6(CLK := output_step_ERR);
bGlobalAuto R= _rt6.Q;

// NETWORK 15
//   bGlobalAuto: Выбор режима Ручной/Авто
_rt7(CLK := output_step_OVER);
IF bGlobalAuto AND NOT output_step_ERR AND NOT output_step_EXEC AND _rt7.Q THEN wStep := input_step_next; END_IF

END_PROGRAM

// MyController/Application/module_unites/MoveTipper_out
PROGRAM MoveTipper_out
VAR_INPUT
	input_step_INIT: BOOL;
	input_step_num: INT;
	input_step_LIM: BOOL;
	input_step_next: INT;
	input_timeout: TIME;
END_VAR

VAR_OUTPUT
	output_step_EXEC: BOOL;
	output_step_OVER: BOOL;
	output_step_ERR: BOOL;
	output_timer_step: TIME;
END_VAR
VAR_IN_OUT
	in_out_ctrl: BOOL;
END_VAR
VAR
	TON_step: TON;
	TON_step_res: BOOL;
	step_active: BOOL;
	TON_delay: TON;
	timer_delay: TIME;
	ton_delay_ok: BOOL;
END_VAR
VAR // added by the converter: edge detectors and wires of the graphical bodies
    _rt1, _rt2, _rt3, _rt4, _rt5, _rt6, _rt7 : R_TRIG;
    _w1, _w2 : BOOL;
    _ft1 : F_TRIG;
END_VAR

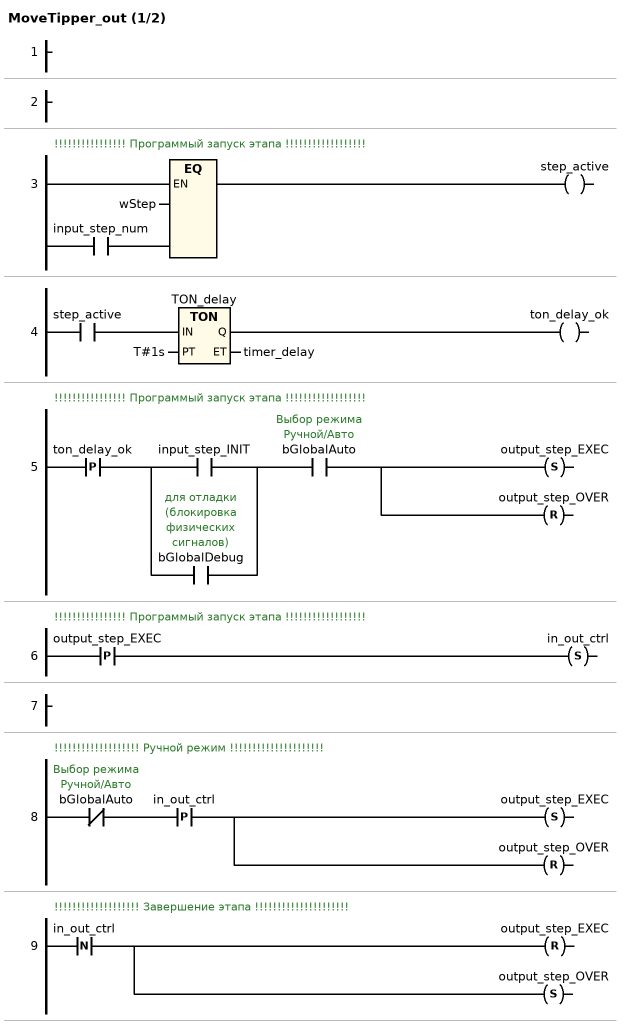
// NETWORK 1

// NETWORK 2

// NETWORK 3
// !!!!!!!!!!!!!!!! Программый запуск этапа !!!!!!!!!!!!!!!!!!
step_active := wStep = input_step_num;

// NETWORK 4
TON_delay(IN := step_active, PT := T#1s, ET => timer_delay); // TON
ton_delay_ok := TON_delay.Q;

// NETWORK 5
// !!!!!!!!!!!!!!!! Программый запуск этапа !!!!!!!!!!!!!!!!!!
//   bGlobalDebug: для отладки (блокировка физических сигналов)
//   bGlobalAuto: Выбор режима Ручной/Авто
_rt1(CLK := ton_delay_ok);
_w1 := _rt1.Q AND (input_step_INIT OR bGlobalDebug) AND bGlobalAuto;
output_step_EXEC S= _w1;
output_step_OVER R= _w1;

// NETWORK 6
// !!!!!!!!!!!!!!!! Программый запуск этапа !!!!!!!!!!!!!!!!!!
_rt2(CLK := output_step_EXEC);
in_out_ctrl S= _rt2.Q;

// NETWORK 7

// NETWORK 8
// !!!!!!!!!!!!!!!!!!! Ручной режим !!!!!!!!!!!!!!!!!!!!!
//   bGlobalAuto: Выбор режима Ручной/Авто
_rt3(CLK := in_out_ctrl);
_w2 := NOT bGlobalAuto AND _rt3.Q;
output_step_EXEC S= _w2;
output_step_OVER R= _w2;

// NETWORK 9
// !!!!!!!!!!!!!!!!!!! Завершение этапа !!!!!!!!!!!!!!!!!!!!!
_ft1(CLK := in_out_ctrl);
output_step_EXEC R= _ft1.Q;
output_step_OVER S= _ft1.Q;

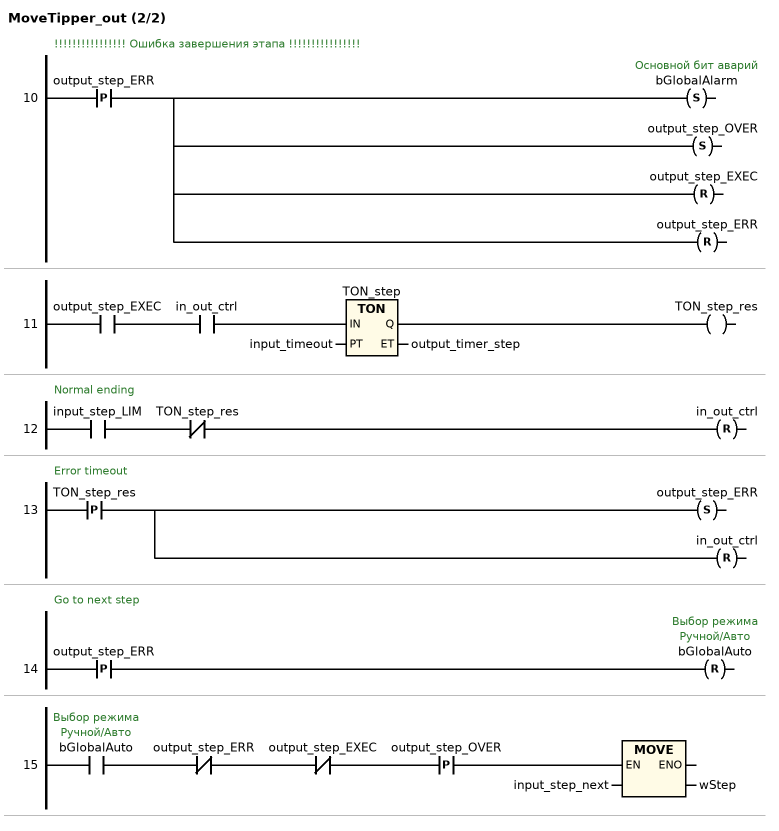
// NETWORK 10
// !!!!!!!!!!!!!!!! Ошибка завершения этапа !!!!!!!!!!!!!!!!
//   bGlobalAlarm: Основной бит аварий
_rt4(CLK := output_step_ERR);
bGlobalAlarm S= _rt4.Q;
output_step_OVER S= _rt4.Q;
output_step_EXEC R= _rt4.Q;
output_step_ERR R= _rt4.Q;

// NETWORK 11
TON_step(IN := output_step_EXEC AND in_out_ctrl, PT := input_timeout, ET => output_timer_step); // TON
TON_step_res := TON_step.Q;

// NETWORK 12
// Normal ending
in_out_ctrl R= input_step_LIM AND NOT TON_step_res;

// NETWORK 13
// Error timeout
_rt5(CLK := TON_step_res);
output_step_ERR S= _rt5.Q;
in_out_ctrl R= _rt5.Q;

// NETWORK 14
// Go to next step
//   bGlobalAuto: Выбор режима Ручной/Авто
_rt6(CLK := output_step_ERR);
bGlobalAuto R= _rt6.Q;

// NETWORK 15
//   bGlobalAuto: Выбор режима Ручной/Авто
_rt7(CLK := output_step_OVER);
IF bGlobalAuto AND NOT output_step_ERR AND NOT output_step_EXEC AND _rt7.Q THEN wStep := input_step_next; END_IF

END_PROGRAM

// MyController/Application/module_unites/FixingFrame_in
PROGRAM FixingFrame_in
VAR_INPUT
	input_step_INIT: BOOL;
	input_step_num: INT;
	input_step_LIM: BOOL;
	input_step_next: INT;
	input_timeout: TIME;
END_VAR

VAR_OUTPUT
	output_step_EXEC: BOOL;
	output_step_OVER: BOOL;
	output_step_ERR: BOOL;
	output_timer_step: TIME;
END_VAR
VAR_IN_OUT
	in_out_ctrl: BOOL;
END_VAR
VAR
	TON_step: TON;
	TON_step_res: BOOL;
	step_active: BOOL;
	TON_delay: TON;
	timer_delay: TIME;
	ton_delay_ok: BOOL;
END_VAR
VAR // added by the converter: edge detectors and wires of the graphical bodies
    _rt1, _rt2, _rt3, _rt4, _rt5, _rt6, _rt7 : R_TRIG;
    _w1, _w2 : BOOL;
    _ft1 : F_TRIG;
END_VAR

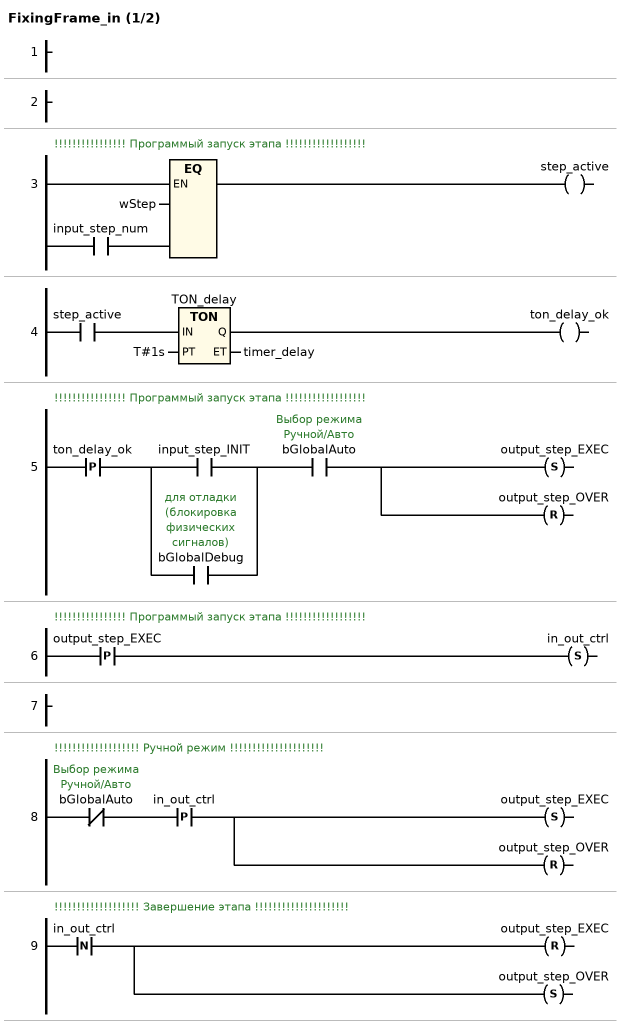
// NETWORK 1

// NETWORK 2

// NETWORK 3
// !!!!!!!!!!!!!!!! Программый запуск этапа !!!!!!!!!!!!!!!!!!
step_active := wStep = input_step_num;

// NETWORK 4
TON_delay(IN := step_active, PT := T#1s, ET => timer_delay); // TON
ton_delay_ok := TON_delay.Q;

// NETWORK 5
// !!!!!!!!!!!!!!!! Программый запуск этапа !!!!!!!!!!!!!!!!!!
//   bGlobalDebug: для отладки (блокировка физических сигналов)
//   bGlobalAuto: Выбор режима Ручной/Авто
_rt1(CLK := ton_delay_ok);
_w1 := _rt1.Q AND (input_step_INIT OR bGlobalDebug) AND bGlobalAuto;
output_step_EXEC S= _w1;
output_step_OVER R= _w1;

// NETWORK 6
// !!!!!!!!!!!!!!!! Программый запуск этапа !!!!!!!!!!!!!!!!!!
_rt2(CLK := output_step_EXEC);
in_out_ctrl S= _rt2.Q;

// NETWORK 7

// NETWORK 8
// !!!!!!!!!!!!!!!!!!! Ручной режим !!!!!!!!!!!!!!!!!!!!!
//   bGlobalAuto: Выбор режима Ручной/Авто
_rt3(CLK := in_out_ctrl);
_w2 := NOT bGlobalAuto AND _rt3.Q;
output_step_EXEC S= _w2;
output_step_OVER R= _w2;

// NETWORK 9
// !!!!!!!!!!!!!!!!!!! Завершение этапа !!!!!!!!!!!!!!!!!!!!!
_ft1(CLK := in_out_ctrl);
output_step_EXEC R= _ft1.Q;
output_step_OVER S= _ft1.Q;

